% RSLogix 500 project P10_KOBIERSKI_M.RSS, saved by version 8.30.00.16 %
PROJECT "UNTITLED"    % processor: Bul.1763 MicroLogix 1100 Series B %

PROGRAM FILES
  LAD 2 "MAIN"  4 rungs
  LAD 3 "IO"  9 rungs
  LAD 4 "CYCLE"  5 rungs
  LAD 5 "CTRL"  14 rungs

DATA FILES
  O0 OUTPUT  4 elements
  I1 INPUT  6 elements
  S2 STATUS  66 elements
  B3 BINARY  2 elements
  T4 TIMER  4 elements
  C5 COUNTER  1 elements
  R6 CONTROL  1 elements
  N7 INTEGER  6 elements
  F8 FLOAT  1 elements

LADDER 2 "MAIN"
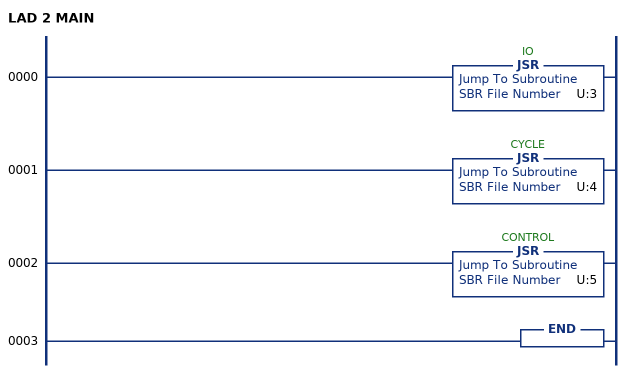
% Rung: 0 %
SOR JSR U:3 EOR
%   U:3  "IO" %
% Rung: 1 %
SOR JSR U:4 EOR
%   U:4  "CYCLE" %
% Rung: 2 %
SOR JSR U:5 EOR
%   U:5  "CONTROL" %
% Rung: 3 %
SOR END EOR

LADDER 3 "IO"
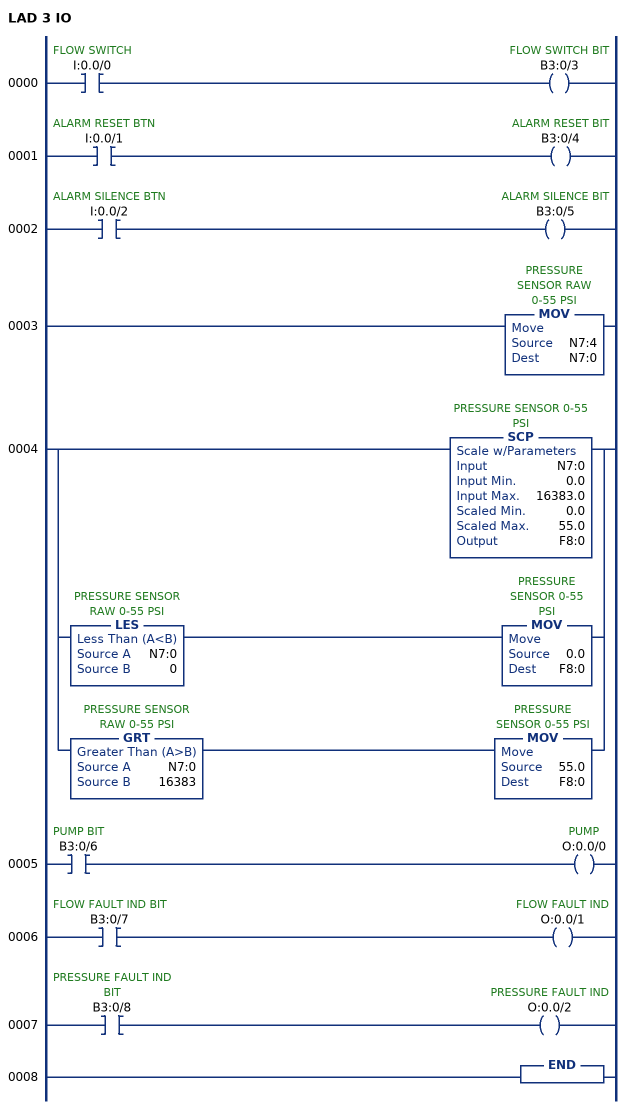
% Rung: 0 %
SOR XIC I:0.0/0 OTE B3:0/3 EOR
%   I:0.0/0  "FLOW SWITCH" %
%   B3:0/3  "FLOW SWITCH BIT" %
% Rung: 1 %
SOR XIC I:0.0/1 OTE B3:0/4 EOR
%   I:0.0/1  "ALARM RESET BTN" %
%   B3:0/4  "ALARM RESET BIT" %
% Rung: 2 %
SOR XIC I:0.0/2 OTE B3:0/5 EOR
%   I:0.0/2  "ALARM SILENCE BTN" %
%   B3:0/5  "ALARM SILENCE BIT" %
% Rung: 3 %
SOR MOV N7:4 N7:0 EOR
%   N7:4  "TEST SET PRESSURE SENSOR PSI" %
%   N7:0  "PRESSURE SENSOR RAW 0-55 PSI" %
% Rung: 4 %
SOR BST SCP N7:0 0.0 16383.0 0.0 55.0 F8:0 NXB LES N7:0 0 MOV 0.0 F8:0 NXB GRT N7:0 16383 MOV 55.0 F8:0 BND EOR
%   N7:0  "PRESSURE SENSOR RAW 0-55 PSI" %
%   F8:0  "PRESSURE SENSOR 0-55 PSI" %
% Rung: 5 %
SOR XIC B3:0/6 OTE O:0.0/0 EOR
%   B3:0/6  "PUMP BIT" %
%   O:0.0/0  "PUMP" %
% Rung: 6 %
SOR XIC B3:0/7 OTE O:0.0/1 EOR
%   B3:0/7  "FLOW FAULT IND BIT" %
%   O:0.0/1  "FLOW FAULT IND" %
% Rung: 7 %
SOR XIC B3:0/8 OTE O:0.0/2 EOR
%   B3:0/8  "PRESSURE FAULT IND BIT" %
%   O:0.0/2  "PRESSURE FAULT IND" %
% Rung: 8 %
SOR END EOR

LADDER 4 "CYCLE"
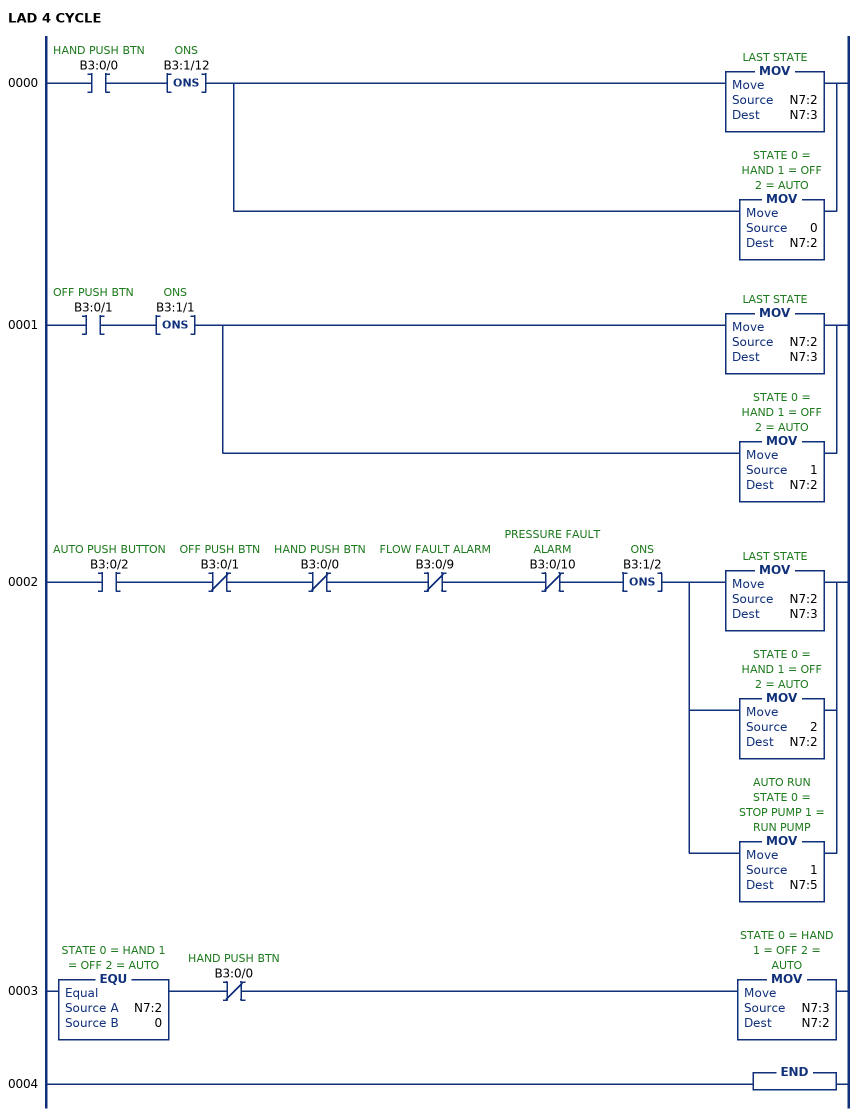
% Rung: 0 %
SOR XIC B3:0/0 ONS B3:1/12 BST MOV N7:2 N7:3 NXB MOV 0 N7:2 BND EOR
%   B3:0/0  "HAND PUSH BTN" %
%   B3:1/12  "ONS" %
%   N7:2  "STATE 0 = HAND 1 = OFF 2 = AUTO" %
%   N7:3  "LAST STATE" %
% Rung: 1 %
SOR XIC B3:0/1 ONS B3:1/1 BST MOV N7:2 N7:3 NXB MOV 1 N7:2 BND EOR
%   B3:0/1  "OFF PUSH BTN" %
%   B3:1/1  "ONS" %
%   N7:2  "STATE 0 = HAND 1 = OFF 2 = AUTO" %
%   N7:3  "LAST STATE" %
% Rung: 2 %
SOR XIC B3:0/2 XIO B3:0/1 XIO B3:0/0 XIO B3:0/9 XIO B3:0/10 ONS B3:1/2 BST MOV N7:2 N7:3 NXB MOV 2 N7:2 NXB MOV 1 N7:5 BND EOR
%   B3:0/2  "AUTO PUSH BUTTON" %
%   B3:0/1  "OFF PUSH BTN" %
%   B3:0/0  "HAND PUSH BTN" %
%   B3:0/9  "FLOW FAULT ALARM" %
%   B3:0/10  "PRESSURE FAULT ALARM" %
%   B3:1/2  "ONS" %
%   N7:2  "STATE 0 = HAND 1 = OFF 2 = AUTO" %
%   N7:3  "LAST STATE" %
%   N7:5  "AUTO RUN STATE 0 = STOP PUMP 1 = RUN PUMP" %
% Rung: 3 %
SOR EQU N7:2 0 XIO B3:0/0 MOV N7:3 N7:2 EOR
%   N7:2  "STATE 0 = HAND 1 = OFF 2 = AUTO" %
%   B3:0/0  "HAND PUSH BTN" %
%   N7:3  "LAST STATE" %
% Rung: 4 %
SOR END EOR

LADDER 5 "CTRL"
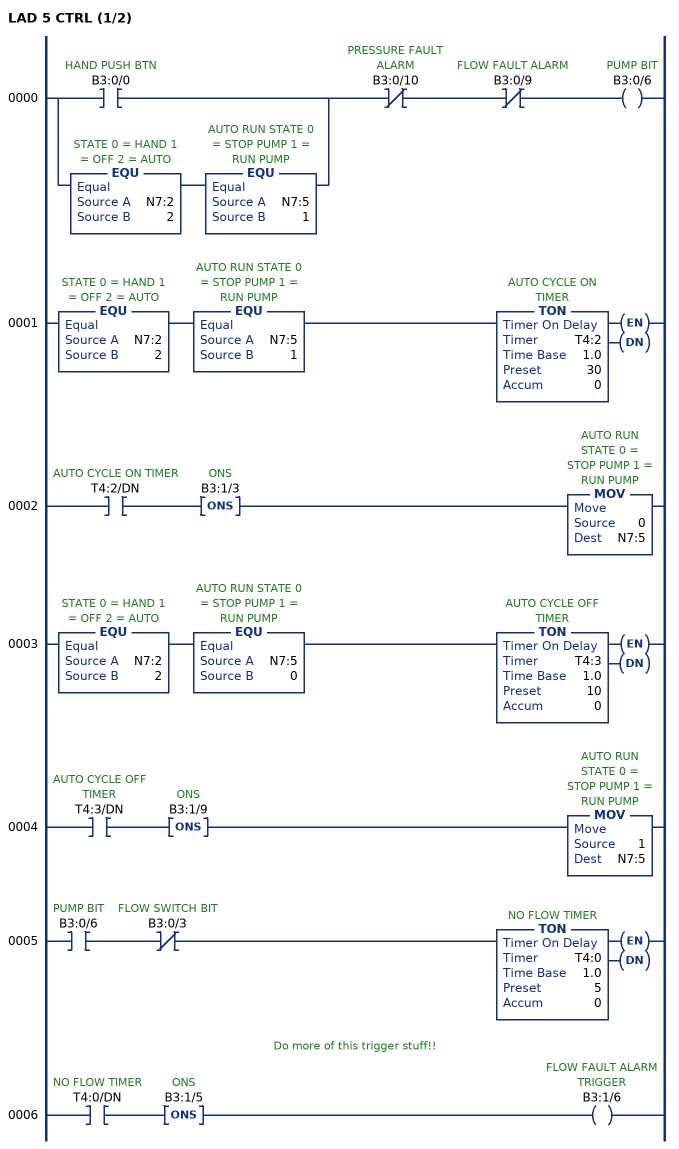
% Rung: 0 %
SOR BST XIC B3:0/0 NXB EQU N7:2 2 EQU N7:5 1 BND XIO B3:0/10 XIO B3:0/9 OTE B3:0/6 EOR
%   B3:0/0  "HAND PUSH BTN" %
%   N7:2  "STATE 0 = HAND 1 = OFF 2 = AUTO" %
%   N7:5  "AUTO RUN STATE 0 = STOP PUMP 1 = RUN PUMP" %
%   B3:0/10  "PRESSURE FAULT ALARM" %
%   B3:0/9  "FLOW FAULT ALARM" %
%   B3:0/6  "PUMP BIT" %
% Rung: 1 %
SOR EQU N7:2 2 EQU N7:5 1 TON T4:2 1.0 30 0 EOR
%   N7:2  "STATE 0 = HAND 1 = OFF 2 = AUTO" %
%   N7:5  "AUTO RUN STATE 0 = STOP PUMP 1 = RUN PUMP" %
%   T4:2  "AUTO CYCLE ON TIMER" %
% Rung: 2 %
SOR XIC T4:2/DN ONS B3:1/3 MOV 0 N7:5 EOR
%   T4:2  "AUTO CYCLE ON TIMER" %
%   B3:1/3  "ONS" %
%   N7:5  "AUTO RUN STATE 0 = STOP PUMP 1 = RUN PUMP" %
% Rung: 3 %
SOR EQU N7:2 2 EQU N7:5 0 TON T4:3 1.0 10 0 EOR
%   N7:2  "STATE 0 = HAND 1 = OFF 2 = AUTO" %
%   N7:5  "AUTO RUN STATE 0 = STOP PUMP 1 = RUN PUMP" %
%   T4:3  "AUTO CYCLE OFF TIMER" %
% Rung: 4 %
SOR XIC T4:3/DN ONS B3:1/9 MOV 1 N7:5 EOR
%   T4:3  "AUTO CYCLE OFF TIMER" %
%   B3:1/9  "ONS" %
%   N7:5  "AUTO RUN STATE 0 = STOP PUMP 1 = RUN PUMP" %
% Rung: 5 %
SOR XIC B3:0/6 XIO B3:0/3 TON T4:0 1.0 5 0 EOR
%   B3:0/6  "PUMP BIT" %
%   B3:0/3  "FLOW SWITCH BIT" %
%   T4:0  "NO FLOW TIMER" %
% Rung: 6 %
% Do more of this trigger stuff!! %
SOR XIC T4:0/DN ONS B3:1/5 OTE B3:1/6 EOR
%   T4:0  "NO FLOW TIMER" %
%   B3:1/5  "ONS" %
%   B3:1/6  "FLOW FAULT ALARM TRIGGER" %

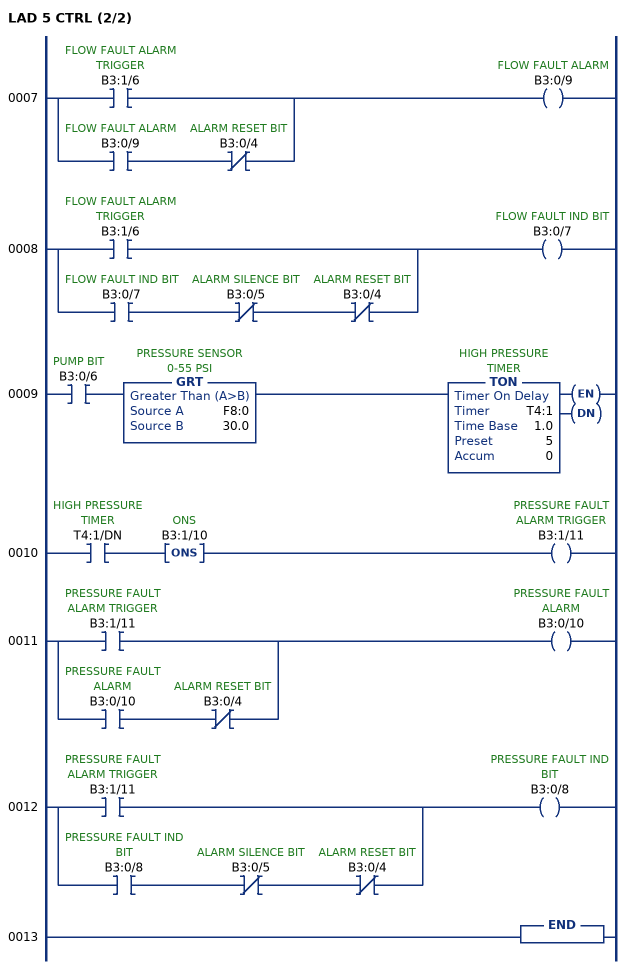
% Rung: 7 %
SOR BST XIC B3:1/6 NXB XIC B3:0/9 XIO B3:0/4 BND OTE B3:0/9 EOR
%   B3:1/6  "FLOW FAULT ALARM TRIGGER" %
%   B3:0/9  "FLOW FAULT ALARM" %
%   B3:0/4  "ALARM RESET BIT" %
% Rung: 8 %
SOR BST XIC B3:1/6 NXB XIC B3:0/7 XIO B3:0/5 XIO B3:0/4 BND OTE B3:0/7 EOR
%   B3:1/6  "FLOW FAULT ALARM TRIGGER" %
%   B3:0/7  "FLOW FAULT IND BIT" %
%   B3:0/5  "ALARM SILENCE BIT" %
%   B3:0/4  "ALARM RESET BIT" %
% Rung: 9 %
SOR XIC B3:0/6 GRT F8:0 30.0 TON T4:1 1.0 5 0 EOR
%   B3:0/6  "PUMP BIT" %
%   F8:0  "PRESSURE SENSOR 0-55 PSI" %
%   T4:1  "HIGH PRESSURE TIMER" %
% Rung: 10 %
SOR XIC T4:1/DN ONS B3:1/10 OTE B3:1/11 EOR
%   T4:1  "HIGH PRESSURE TIMER" %
%   B3:1/10  "ONS" %
%   B3:1/11  "PRESSURE FAULT ALARM TRIGGER" %
% Rung: 11 %
SOR BST XIC B3:1/11 NXB XIC B3:0/10 XIO B3:0/4 BND OTE B3:0/10 EOR
%   B3:1/11  "PRESSURE FAULT ALARM TRIGGER" %
%   B3:0/10  "PRESSURE FAULT ALARM" %
%   B3:0/4  "ALARM RESET BIT" %
% Rung: 12 %
SOR BST XIC B3:1/11 NXB XIC B3:0/8 XIO B3:0/5 XIO B3:0/4 BND OTE B3:0/8 EOR
%   B3:1/11  "PRESSURE FAULT ALARM TRIGGER" %
%   B3:0/8  "PRESSURE FAULT IND BIT" %
%   B3:0/5  "ALARM SILENCE BIT" %
%   B3:0/4  "ALARM RESET BIT" %
% Rung: 13 %
SOR END EOR

OTHER DOCUMENTED ADDRESSES
  B3:0/11  "SYSTEM ON"
  B3:1/0  "ONS"
  B3:1/4  "AUTO RUN BIT"
  B3:1/7  "ONS"
  B3:1/8  "PRESSURE FAULT ALARM TRIGGER"
  N7:1  "PRESSURE SENSOR 0-55 PSI"

DATA TABLE (non-zero values as saved)
DATA T4
% .PRE .ACC %
% T4:0 % 5 0
% T4:1 % 5 0
% T4:2 % 30 0
% T4:3 % 10 0
DATA N7
% N7:0 % 0 0 0 0 40 0
DATA F8
% F8:0 % 33.57138
